INTERFACE ITF_GroupElement

END_INTERFACE

(* stored: Version 1.1.0.1, ProductVersion 3.1.4024.15
   Itf ITF_GroupElement: Id {5227295f-e3f4-478a-9ab8-5c8a8c15e80d} *)
